INTERFACE IGuard

PROPERTY direction : Rotation
GET
END_GET
SET
END_SET
END_PROPERTY

METHOD walk
VAR_INPUT
	map :I2dArray;
END_VAR
END_METHOD

PROPERTY x : DINT
GET
END_GET
SET
END_SET
END_PROPERTY

PROPERTY y : DINT
GET
END_GET
SET
END_SET
END_PROPERTY

END_INTERFACE

(* stored: Version 1.1.0.1
   Itf IGuard: Id {f2b2b829-faf3-4b6e-b1b8-c13d026452dc}
   Property direction: Id {b8254941-eba0-4810-986b-5e372dc9e805}
   Get Get: Id {f3a21c21-f7d3-4b12-99f2-709f0fac04b7}
   Set Set: Id {1b429841-f5b8-421a-8e7b-16c2d35a940f}
   Method walk: Id {6f02a1d2-f5e9-436f-bf4e-74f98c745008}
   Property x: Id {1f1f695e-9310-48bf-a85b-ebda0d43e411}
   Get Get: Id {fba93a85-e7c3-4c8a-be66-15bd7d9b23ec}
   Set Set: Id {4c2f2195-acc6-4ae8-8551-f75417517614}
   Property y: Id {a413a7c4-99f4-4fef-a5f0-e81f28a124e5}
   Get Get: Id {e40c0bc4-6c59-4908-8f19-fae4d482ba5a}
   Set Set: Id {bb6eb65f-6e97-4733-81f5-ae2d7c3d12f0} *)
